PROGRAM p_MPSSup
VAR
END_VAR


q_xXCS_MPSOK := g_xIOState AND vgcPBT_VGC_01.i_xOpnLS AND vgcPBT_VGC_02.i_xOpnLS AND vgcPBT_VGC_03.i_xOpnLS AND vgcPBT_VGC_04.i_xOpnLS;
//

END_PROGRAM

(* stored: Version 1.1.0.1, ProductVersion 3.1.4020.12
   POU p_MPSSup: Id {606dda39-341f-4609-835a-4778708a8932}, SpecialFunc None *)
